FUNCTION_BLOCK StepChain_1
VAR_INPUT
END_VAR
VAR_OUTPUT
END_VAR
VAR
	fbSynchPayload : SynchPayload;
	step : UINT;
END_VAR

CASE step OF
	
	0:
		IF 	fbPayloadCarrier
				.SetPayload(
					fbSynchPayload,
					SYNCH_PAYLOAD,
					ONE_TO_ONE,
					THIS
				)	
			THEN
			
			step := 10;
		END_IF
		
	10:
	
		fbSynchPayload.bReleaseRequest := TRUE;
		IF 	fbSynchPayload.bReleaseRequestReceived
			THEN
			fbSynchPayload.bReleaseRequest := FALSE;
			step := 20;
		END_IF
		
	20:
		IF  fbSynchPayload.bRequestAck
			THEN
			fbSynchPayload.bRequestAckReceived := TRUE;
			step := 30;
		END_IF
		
	30:	

		fbSynchPayload.bRequestAckReceived := FALSE;
		step := 40;
		
	40:
	
		fbPayloadCarrier.ResetPayload(THIS);
		step := 50;
		
		
END_CASE

END_FUNCTION_BLOCK

(* stored: Version 1.1.0.1, ProductVersion 3.1.4024.2
   POU StepChain_1: Id {f737c90b-0d93-4659-9531-9886105b95f1}, SpecialFunc None *)
